// TwinCAT 3 PLC project PlcMotor
// ProgramVersion: 3.1.4024.0
// project tree:
//   POUs/ FB_Motor.TcPOU, MAIN.TcPOU

// ---- POUs/FB_Motor.TcPOU
FUNCTION_BLOCK FB_Motor
VAR
    speed : REAL;
END_VAR

METHOD SetSpeed
VAR_INPUT
    value : REAL;
END_VAR
speed := value;
END_METHOD

METHOD Stop
END_METHOD

END_FUNCTION_BLOCK

// ---- POUs/MAIN.TcPOU
PROGRAM MAIN
VAR
    motor : FB_Motor;
END_VAR

motor.SetSpeed(value := 1.0);
motor.Stop();

END_PROGRAM
